{attribute 'GeneratedUsingTerminal: DL-EC1A-0000'}
{attribute addProperty BoxType "DL-EC1A-0000"}
{attribute addProperty Id "AdsAddrAT %I*AMSADDR8StateAT %I*UINT2"}
{attribute addProperty CRC "854291690"}
{attribute addProperty Size "10"}
TYPE
    InfoData EXTENDS InputBase_8311D824 :
    STRUCT
        {attribute addProperty Name "AdsAddr"}
        AdsAddr AT %I* : AMSADDR;
        {attribute addProperty Name "State"}
        State AT %I* : UINT;
    END_STRUCT
END_TYPE

(* stored: Version 1.1.0.1, ProductVersion 3.1.4024.12
   DUT InfoData: Id {b41ac276-a724-055d-027f-b1267238c302} *)
